Staubli VAL3: iFluorClosed.pgx

public program iFluorClosed(num& nNum[] (dimensions=1))
begin
  nNum=dioGet(iFluorClosed)
end
